FUNCTION_BLOCK FB_FDM_EL2521_Ref EXTENDS FB_ExtruderRef
VAR_INPUT
END_VAR
VAR
	pPTOStepperRef : POINTER TO ST_PTOStepperRef;
END_VAR
VAR_OUTPUT
	
END_VAR

METHOD FB_init : BOOL
VAR_INPUT
	bInitRetains : BOOL; // if TRUE, the retain variables are initialized (warm start / cold start)
	bInCopyCode : BOOL;  // if TRUE, the instance afterwards gets moved into the copy code (online change)
	stPTOStepperRef : POINTER TO ST_PTOStepperRef;
END_VAR
THIS^.pPTOStepperRef := stPTOStepperRef;
END_METHOD

PROPERTY P_bError : BOOL
GET
END_GET
END_PROPERTY

PROPERTY P_bIsActive : BOOL
GET
END_GET
END_PROPERTY

PROPERTY P_bIsLocked : BOOL
GET
P_bIsLocked := TRUE;
END_GET
END_PROPERTY

PROPERTY P_pPTOStepperRef : POINTER TO ST_PTOStepperRef
GET
P_pPTOStepperRef := pPTOStepperRef;
END_GET
END_PROPERTY

END_FUNCTION_BLOCK

(* stored: Version 1.1.0.1, ProductVersion 3.1.4024.11
   POU FB_FDM_EL2521_Ref: Id {d33781aa-cc03-4ae1-a1d7-a4f6e7c69809}, SpecialFunc None
   Method FB_init: Id {a4e05b4b-3e29-430d-ba87-1d09854bf17a}
   Property P_bError: Id {af83d4f0-e2c3-4940-89b2-c323f3f0134d}
   Get Get: Id {6b8ecbd2-526b-4fff-82ce-dc98ecb26531}
   Property P_bIsActive: Id {e44f5898-4601-438a-93b7-1eaea22c632e}
   Get Get: Id {02f127e9-9235-4e28-a2b9-47a94a42d4a3}
   Property P_bIsLocked: Id {74c5c070-ab90-4b41-8988-b6a5b9fb2bb6}
   Get Get: Id {5a27fea1-6fd2-4b3c-bcec-f00b63eb67bc}
   Property P_pPTOStepperRef: Id {7c395262-d7b9-44d7-8bf1-9ff017ae7882}
   Get Get: Id {bfa401f1-0340-4f32-808d-22a8eaffe8a9} *)
